FUNCTION alg_M_Distributing_pickpos : ARRAY[0..3] OF DINT
VAR_INPUT
	state: STATE;
END_VAR

alg_M_Distributing_pickpos := makeArray0(0, 1, 0, 2);

END_FUNCTION

(* stored: Version 1.1.0.1, ProductVersion 3.1.4022.18
   POU alg_M_Distributing_pickpos: Id {a4a658ff-196c-494a-9af6-c9f0e7b93851}, SpecialFunc None *)
